VAR_GLOBAL
END_VAR

(* stored: Version 1.1.0.1, ProductVersion 3.1.4024.11
   GVL OP50_Recipe: Id {869f193b-cec0-48e9-833e-675858802209} *)
